(* IEC 61131-3 sources: Lasal/CPU_5344_V01/Class/sLineHandler, 1 file *)

(* ---- sLineHandler.st ---- *)
(*!
<Class
	Name               = "sLineHandler"
	Revision           = "1.0"
	RealtimeTask       = "false"
	CyclicTask         = "true"
	DefCyclictime      = "10 ms"
	BackgroundTask     = "false"
	Sigmatek           = "false"
	OSInterface        = "false"
	HighPriority       = "false"
	Automatic          = "false"
	UpdateMode         = "Prescan"
	SharedCommandTable = "true"
	Objectsize         = "(1140,1440)">
	<Channels>
		<Server Name="actLengthInInput" Visualized="true" Initialize="false" WriteProtected="false" Retentive="false"/>
		<Server Name="actMathHeigth" Visualized="true" Initialize="false" WriteProtected="false" Retentive="false"/>
		<Server Name="actMathWidth" Visualized="true" Initialize="false" WriteProtected="false" Retentive="false"/>
		<Server Name="amountDone" Visualized="true" Initialize="false" WriteProtected="false" Retentive="false"/>
		<Server Name="amountToDo" Visualized="true" Initialize="false" WriteProtected="false" Retentive="false"/>
		<Server Name="BackOffMaterial" Visualized="true" Initialize="false" WriteProtected="false" Retentive="false"/>
		<Server Name="ClassSvr" Visualized="false" Initialize="false" WriteProtected="true" Retentive="false"/>
		<Server Name="FrontOffMaterial" Visualized="true" Initialize="false" WriteProtected="false" Retentive="false"/>
		<Server Name="lineNrInput" Visualized="true" Initialize="false" WriteProtected="false" Retentive="false"/>
		<Server Name="lineNrOutput" Visualized="true" Initialize="false" WriteProtected="false" Retentive="false"/>
		<Server Name="reReadAmountToDo" Visualized="true" Initialize="false" WriteProtected="false" Retentive="false"/>
		<Server Name="ResetBackOffMaterial" Visualized="true" Initialize="false" WriteProtected="false" Retentive="false"/>
		<Server Name="ResetFrontOffMaterialToTakeIn" Visualized="false" Initialize="false" WriteProtected="false" Retentive="false"/>
		<Server Name="rnrInput" Visualized="false" Initialize="false" WriteProtected="false" Retentive="false"/>
		<Server Name="rnrOutput" Visualized="false" Initialize="false" WriteProtected="false" Retentive="false"/>
		<Server Name="sSetBackOffMaterialAfterSawing" Visualized="false" Initialize="true" DefValue="1" WriteProtected="true" Retentive="false"/>
		<Server Name="stopAfterLength" Visualized="true" Initialize="false" WriteProtected="false" Retentive="false"/>
		<Server Name="stprInputSide" Visualized="true" Initialize="false" WriteProtected="false" Retentive="false"/>
		<Server Name="stprOutputSide" Visualized="true" Initialize="false" WriteProtected="false" Retentive="false"/>
		<Server Name="stsCompleted" Visualized="false" Initialize="false" WriteProtected="true" Retentive="false"/>
		<Server Name="stsStartedFromPC" Visualized="false" Initialize="false" WriteProtected="false" Retentive="false"/>
		<Server Name="thisUnitIsSaw" Visualized="false" Initialize="true" DefValue="1" WriteProtected="true" Retentive="false"/>
		<Client Name="ctrlMain" Required="true" Internal="false"/>
		<Client Name="ctrlReadIn" Required="true" Internal="false"/>
		<Client Name="iActMathHeigth" Required="true" Internal="false"/>
		<Client Name="iActMathWidth" Required="true" Internal="false"/>
		<Client Name="iAmountToDo" Required="true" Internal="false"/>
		<Client Name="iInputLength" Required="true" Internal="false"/>
		<Client Name="iLiveXPos" Required="true" Internal="false"/>
		<Client Name="iOffsetInputMaterial" Required="true" Internal="false"/>
		<Client Name="listSLines" Required="true" Internal="false"/>
		<Client Name="oAmountDone" Required="true" Internal="false"/>
		<Client Name="oAmountDoneOutput" Required="false" Internal="false"/>
		<Client Name="oLineNrInput" Required="true" Internal="false"/>
		<Client Name="oLineNrOutput" Required="true" Internal="false"/>
	</Channels>
</Class>
*)
sLineHandler : CLASS
  //Servers:
	ClassSvr 	: SvrChCmd_DINT;
	stsCompleted 	: SvrCh_DINT;
	stsStartedFromPC 	: SvrCh_DINT;
	stprInputSide 	: SvrCh_DINT;
	stprOutputSide 	: SvrCh_DINT;
	FrontOffMaterial 	: SvrCh_DINT;
	BackOffMaterial 	: SvrCh_DINT;
	ResetBackOffMaterial 	: SvrCh_DINT;
	ResetFrontOffMaterialToTakeIn 	: SvrCh_DINT;
	actLengthInInput 	: SvrCh_DINT;
	actMathHeigth 	: SvrCh_DINT;
	actMathWidth 	: SvrCh_DINT;
	lineNrInput 	: SvrCh_DINT;
	lineNrOutput 	: SvrCh_DINT;
	stopAfterLength 	: SvrCh_DINT;
	amountToDo 	: SvrCh_DINT;
	amountDone 	: SvrCh_DINT;
	reReadAmountToDo 	: SvrCh_DINT;
	thisUnitIsSaw 	: SvrCh_Units;
	sSetBackOffMaterialAfterSawing 	: SvrCh_DINT;
	rnrInput 	: SvrCh_DINT;
	rnrOutput 	: SvrCh_DINT;
  //Clients:
	listSLines 	: CltChCmd_GlobalList;
	ctrlMain 	: CltChCmd_mainControl;
	iInputLength 	: CltCh_DINT;
	iAmountToDo 	: CltCh_DINT;
	iOffsetInputMaterial 	: CltCh_DINT;
	iLiveXPos 	: CltCh_DINT;
	iActMathWidth 	: CltCh_DINT;
	iActMathHeigth 	: CltCh_DINT;
	oAmountDone 	: CltCh_DINT;
	oAmountDoneOutput 	: CltCh_DINT;
	oLineNrInput 	: CltCh_DINT;
	oLineNrOutput 	: CltCh_DINT;
	ctrlReadIn 	: CltChCmd_readInGlobalList;
  //Variables:
		actInputLine 	: SRegelInfo;
		actOutputLine 	: SRegelInfo;
		firstStart 	: DINT;
		lastFrontPosDuringSawing 	: DINT;
  //Functions:

	FUNCTION VIRTUAL GLOBAL CyWork
		VAR_INPUT
			EAX 	: UDINT;
		END_VAR
		VAR_OUTPUT
			state (EAX) 	: UDINT := READY;
		END_VAR;

	FUNCTION GLOBAL startProgram
		VAR_INPUT
			LineNrInput2 	: DINT;
		END_VAR;

	FUNCTION GLOBAL stopProgram;

	FUNCTION stepperInput;

	FUNCTION stepperOutput;

	FUNCTION VIRTUAL GLOBAL ResetBackOffMaterial::Write
		VAR_INPUT
			input (EAX) 	: DINT;
		END_VAR
		VAR_OUTPUT
			result (EAX) 	: DINT;
		END_VAR;

	FUNCTION VIRTUAL GLOBAL ResetFrontOffMaterialToTakeIn::Write
		VAR_INPUT
			input (EAX) 	: DINT;
		END_VAR
		VAR_OUTPUT
			result (EAX) 	: DINT;
		END_VAR;

	FUNCTION VIRTUAL GLOBAL actMathHeigth::Read
		VAR_OUTPUT
			output (EAX) 	: DINT;
		END_VAR;

	FUNCTION VIRTUAL GLOBAL reReadAmountToDo::Write
		VAR_INPUT
			input (EAX) 	: DINT;
		END_VAR
		VAR_OUTPUT
			result (EAX) 	: DINT;
		END_VAR;

	FUNCTION VIRTUAL GLOBAL rnrInput::Write
		VAR_INPUT
			input (EAX) 	: DINT;
		END_VAR
		VAR_OUTPUT
			result (EAX) 	: DINT;
		END_VAR;

	FUNCTION VIRTUAL GLOBAL rnrOutput::Write
		VAR_INPUT
			input (EAX) 	: DINT;
		END_VAR
		VAR_OUTPUT
			result (EAX) 	: DINT;
		END_VAR;
  //Tables:
	FUNCTION @STD
		VAR_OUTPUT
			ret_code	: CONFSTATES;
		END_VAR;
	FUNCTION GLOBAL TAB @CT_;
END_CLASS;

#pragma usingLtd GlobalList
#pragma usingLtd mainControl
#pragma usingLtd readInGlobalList

// JdK 20-6-2019: sLineHandler created for 4284 TraffiRoad. Goal is to handle the s lines for the units
// just run all the sLinerules from begin to end

FUNCTION VIRTUAL GLOBAL sLineHandler::reReadAmountToDo::Write
	VAR_INPUT
		input (EAX) 	: DINT;
	END_VAR
	VAR_OUTPUT
		result (EAX) 	: DINT;
	END_VAR

	reReadAmountToDo := input;
  iAmountToDo:=iAmountToDo.Read();
  amountToDo:=iAmountToDo;
	result := reReadAmountToDo;

END_FUNCTION

FUNCTION GLOBAL sLineHandler::startProgram
	VAR_INPUT
		LineNrInput2 	: DINT;
	END_VAR

  //set everything right for starting
  IF stprInputSide= 0 THEN
    stsCompleted:=0;
    lineNrInput:=LineNrInput2;//0;
    lineNrOutput:=0;
    iInputLength:=iInputLength.Read();
    FrontOffMaterial:=FAULTVALUE; //on start there should be no material, so set values on fault value else we can't possible not start (doesn't fit then)
    BackOffMaterial:=-1*FAULTVALUE;
    oAmountDone:=oAmountDone.Read(); //at start, read in amount already done
    oAmountDoneOutput:=oAmountDone;
    IF stsStartedFromPC= 0 THEN
      amountDone:=oAmountDone;
    ELSE
      amountDone:=0;
    END_IF;
    firstStart:=1;
    stprInputSide:=1;
  END_IF;

END_FUNCTION

FUNCTION GLOBAL sLineHandler::stopProgram

  //just stop it
  stprInputSide:=0;
  stprOutputSide:=0;
  stsCompleted:= 0;

END_FUNCTION

FUNCTION sLineHandler::stepperInput

  CASE stprInputSide OF

  0: //wait
    stsCompleted:= 0;

  1: //take next sLine
    actInputLine:=listSLines.readLine(Nr:=lineNrInput);
    IF actInputLine.Units.DoWithOutput= 0 THEN //check if we have to do this line with the input
      oLineNrInput:=actInputLine.Rnr;
      oLineNrInput.Write(input:=oLineNrInput);
      rnrInput:=oLineNrInput;
      stprInputSide+= 1;
    ELSE
      IF actInputLine.Command= STARTOUTPUT THEN //start working with output, but only if outputstepper is 0
        IF stprOutputSide= 0 THEN
          BackOffMaterial:=0; //for 4255 taking away material with output is always from sawing pos
          lineNrOutput:=lineNrInput+1;
          lineNrInput+= 1;
          stprOutputSide:=1;
        END_IF;
      ELSE
        lineNrInput+=1; //just ignore this rule, because it's for the output
      END_IF;
    END_IF;

  2: //do line action
    CASE actInputLine.Command OF

    STARTCOM: //reset act length input, if first start, read in to do and from line
      IF stsStartedFromPC= 0 THEN
        actLengthInInput:=iInputLength;
        iActMathHeigth:= iActMathHeigth.Read(); //JdK 29-9-2020: should go through sline list, but isn't ready yet
        iActMathWidth:= iActMathWidth.Read();
        actMathHeigth:= iActMathHeigth;
        actMathWidth:= iActMathWidth;
      ELSE
        actLengthInInput:= ctrlReadIn.stsActInputLength;
        actMathHeigth:= ctrlReadIn.stsActInputHeigth;
        actMathWidth:= ctrlReadIn.stsActInputWidth;
      END_IF;

      IF firstStart=1 THEN
        amountToDo:=actInputLine.Amount;
        firstStart:=0;
      END_IF;
      stprInputSide:=5;

    STOPCOM:
      amountDone+=1;
      IF stsStartedFromPC= 0 THEN
        oAmountDone+=1; //one extra ready
        oAmountDone.Write(input:=oAmountDone);
      END_IF;
      FrontOffMaterial:= FAULTVALUE; //ready with production on input, so reset front off material
      lineNrInput:=-1; //because in stpr 5 value 1 is added
      IF stopAfterLength= 1 THEN
        stprInputSide:= 10; //wait there until output is ready, but after restart we can go on
        stopAfterLength:= 0;
      ELSIF amountDone >= amountToDo THEN //amount reached
        IF stsStartedFromPC= 0 THEN
          stprInputSide:= 20; //JdK 7-10-2020 only do one assembly 15; //check if we can produce next assembly
        ELSE
          stprInputSide:= 12; //check if we have to do next profile
        END_IF;
      ELSE
        stprInputSide:=5;
      END_IF;

    WAITOPERATIONCOM, WAITFOROUTPUT:
      stprInputSide+= 1;

    UNITMOVECOM, UNITSTARTCOM, CHANGETOOL:
      IF ctrlMain.startSLine(sLine:=actInputLine)= 1 THEN //just start it until we get a 1 back
        IF (actInputLine.Units AND thisUnitIsSaw)>0 & actInputLine.Command= UNITSTARTCOM THEN //means sawing is started
          lastFrontPosDuringSawing:= FrontOffMaterial;
          FrontOffMaterial:=0; //because sawing is done
          IF sSetBackOffMaterialAfterSawing= 1 & stprOutputSide= 0 THEN //for machines without outputrules, set back of material right after sawing
            BackOffMaterial:= 0;
          END_IF;
          iLiveXPos:=iLiveXPos.Read();
          actLengthInInput:= iLiveXPos;
        END_IF;
        stprInputSide:=5;
      ELSE
        //give alarm? started action at wrong time or started not existed unit
      END_IF;

    ELSE
      //give alarm for not possible command

    END_CASE;

  3: //wait actions
    IF actInputLine.Command= WAITOPERATIONCOM THEN
      IF ctrlMain.askReadySLine(sLine:=actInputLine)= 1 THEN //wait until we get back a ready
        stprInputSide:=5;
      END_IF;
    ELSIF actInputLine.Command= WAITFOROUTPUT THEN
      IF stprOutputSide= 0 THEN //just wait until output is done
        stprInputSide:=5;
      END_IF;
    END_IF;

  5: //prepare for next line
    lineNrInput+=1;
    stprInputSide:= 1;

  10: //stop after length place, wait until output done
    IF stprOutputSide= 0 THEN
      stprInputSide+=1;
    END_IF;

  11: //after main puts machine in hold (also in and output), main also sets stpr input to 5

  12: //check if we have to do next program in list (started from pc)

  13: //just wait

  14: //restart with next line
    lineNrInput:= 0;
    stprInputSide:= 1;

  15: //wait until output is done
    IF stprOutputSide= 0 THEN
      stprInputSide+= 1;
    END_IF;

  16: //write next recipeid to assembly
    //ctrlAssembly.RecipeId.Write(input:=ctrlAssembly.RecipeId+1);
    iAmountToDo:= iAmountToDo.Read();
    oAmountDone:= oAmountDone.Read();
    iInputLength:= iInputLength.Read();
    IF iAmountToDo > oAmountDone & iInputLength > 0 THEN
      ctrlMain.calcNext();
      stprInputSide:= 0;
    ELSE
      stprInputSide:= 20; //next is also empty, so stop it
    END_IF;

  17: //step after stopped after length
    IF amountDone >= amountToDo THEN //amount reached
      IF stsStartedFromPC= 0 THEN
        stprInputSide:= 15; //check if we can produce next assembly
      ELSE
        stprInputSide:= 12; //check if we have to do next profile
      END_IF;
    ELSE
      stprInputSide:=5;
    END_IF;

  20: //wait until output is done
    IF stprOutputSide= 0 THEN
      stprInputSide+= 1;
    END_IF;

  21: //give ready signal, stop is done by main
    stsCompleted:=1;

  END_CASE;

END_FUNCTION

FUNCTION sLineHandler::stepperOutput

  CASE stprOutputSide OF

  0: //just wait

  1: //get new line
    actOutputLine:= listSLines.readLine(Nr:=lineNrOutput);
    IF actOutputLine.Units.DoWithOutput= 1 THEN
      oLineNrOutput:= lineNrOutput;
      oLineNrOutput.Write(input:=oLineNrOutput);
      rnrOutput:=oLineNrOutput;
      stprOutputSide+=1;
    ELSE
      lineNrOutput+= 1;
    END_IF;

  2: //do line action
    CASE actOutputLine.Command OF

    STARTCOM: //should not happen for output
      stprOutputSide:=5; //just ignore

    STOPCOM: //do counting and ready, counting is discussion, is it the only stopcom for this product?
      oAmountDoneOutput+=1;
      oAmountDoneOutput.Write(input:=oAmountDoneOutput);
      //dont reset backside, because material can still be somewehere on the outputlane
      lineNrOutput:=0;
      stprOutputSide:=0; //after stopcom, just stop

    WAITOPERATIONCOM:
      stprOutputSide+= 1;

    UNITMOVECOM, UNITSTARTCOM, CHANGETOOL:
      IF ctrlMain.startSLine(sLine:=actOutputLine)= 1 THEN //just start it until we get a 1 back
        stprOutputSide:=5;
      ELSE
        //give alarm? started action at wrong time or started not existed unit
      END_IF;

    ELSE
      //give alarm for not possible command

    END_CASE;

  3: //waiting action, for output should only be wait operation
    IF actOutputLine.Command= WAITOPERATIONCOM THEN
      IF ctrlMain.askReadySLine(sLine:=actOutputLine)= 1 THEN //wait until we get back a ready
        stprOutputSide:=5;
      END_IF;
    END_IF;

  5: //prepare for next line
    lineNrOutput+=1;
    stprOutputSide:= 1;

  END_CASE;

END_FUNCTION

FUNCTION VIRTUAL GLOBAL sLineHandler::CyWork
	VAR_INPUT
		EAX 	: UDINT;
	END_VAR
	VAR_OUTPUT
		state (EAX) 	: UDINT;(* := READY *)
	END_VAR

  stepperInput();
  stepperOutput();

END_FUNCTION

FUNCTION VIRTUAL GLOBAL sLineHandler::ResetFrontOffMaterialToTakeIn::Write
	VAR_INPUT
		input (EAX) 	: DINT;
	END_VAR
	VAR_OUTPUT
		result (EAX) 	: DINT;
	END_VAR

  //after take in new material, we have to reset front to offset of input
	ResetFrontOffMaterialToTakeIn := input;
  iOffsetInputMaterial:=iOffsetInputMaterial.Read();
  FrontOffMaterial:=iOffsetInputMaterial;
	result := ResetFrontOffMaterialToTakeIn;

END_FUNCTION

FUNCTION VIRTUAL GLOBAL sLineHandler::ResetBackOffMaterial::Write
	VAR_INPUT
		input (EAX) 	: DINT;
	END_VAR
	VAR_OUTPUT
		result (EAX) 	: DINT;
	END_VAR

	ResetBackOffMaterial := input;
  BackOffMaterial:=ResetBackOffMaterial;
	result := ResetBackOffMaterial;

END_FUNCTION

FUNCTION VIRTUAL GLOBAL sLineHandler::actMathHeigth::Read
	VAR_OUTPUT
		output (EAX) 	: DINT;
	END_VAR

  iActMathHeigth:= iActMathHeigth.Read(); //temp solution, should come from calclist
  //actMathHeigth:= iActMathHeigth;
	output := actMathHeigth;

END_FUNCTION

FUNCTION VIRTUAL GLOBAL sLineHandler::rnrInput::Write
	VAR_INPUT
		input (EAX) 	: DINT;
	END_VAR
	VAR_OUTPUT
		result (EAX) 	: DINT;
	END_VAR

	rnrInput := input;
  oLineNrInput:=rnrInput;
  oLineNrInput.Write(input:=oLineNrInput);
	result := rnrInput;

END_FUNCTION

FUNCTION VIRTUAL GLOBAL sLineHandler::rnrOutput::Write
	VAR_INPUT
		input (EAX) 	: DINT;
	END_VAR
	VAR_OUTPUT
		result (EAX) 	: DINT;
	END_VAR

	rnrOutput := input;
  oLineNrOutput:=rnrOutput;
  oLineNrOutput.Write(input:=oLineNrOutput);
	result := rnrOutput;

END_FUNCTION
